// TIA Portal V17 export
// export: Created 2021-12-03T08:13:14.6576163Z, ExportSetting WithDefaults, DisplayName Totally Integrated Automation Portal, DisplayVersion V17, DisplayName TIA Portal Openness, DisplayVersion V17, DisplayName TIA Portal Version Control Interface, DisplayVersion V17, DisplayName STEP 7 Professional, DisplayVersion V17, DisplayName STEP 7 Safety, DisplayVersion V17, DisplayName WinCC Advanced, DisplayVersion V17
FUNCTION "FFC_ReadInputs" : Void   // FC50, F_FBD
VERSION : 0.1
// stored: AutoNumber false, IsIECCheckEnabled false, UDAEnableTagReadback false
BEGIN

REGION Network 2: Консоль ускорителя канал 1
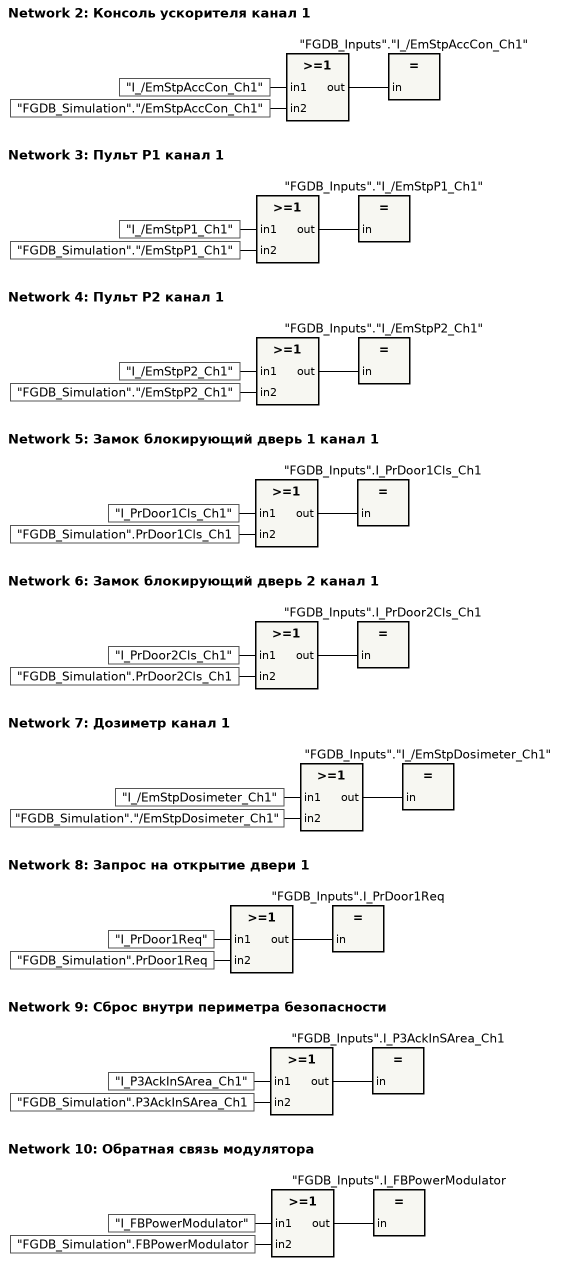
   "FGDB_Inputs"."I_/EmStpAccCon_Ch1" := "I_/EmStpAccCon_Ch1" OR "FGDB_Simulation"."/EmStpAccCon_Ch1";
END_REGION

REGION Network 3: Пульт Р1 канал 1
   "FGDB_Inputs"."I_/EmStpP1_Ch1" := "I_/EmStpP1_Ch1" OR "FGDB_Simulation"."/EmStpP1_Ch1";
END_REGION

REGION Network 4: Пульт Р2 канал 1
   "FGDB_Inputs"."I_/EmStpP2_Ch1" := "I_/EmStpP2_Ch1" OR "FGDB_Simulation"."/EmStpP2_Ch1";
END_REGION

REGION Network 5: Замок блокирующий дверь 1 канал 1
   "FGDB_Inputs".I_PrDoor1Cls_Ch1 := "I_PrDoor1Cls_Ch1" OR "FGDB_Simulation".PrDoor1Cls_Ch1;
END_REGION

REGION Network 6: Замок блокирующий дверь 2 канал 1
   "FGDB_Inputs".I_PrDoor2Cls_Ch1 := "I_PrDoor2Cls_Ch1" OR "FGDB_Simulation".PrDoor2Cls_Ch1;
END_REGION

REGION Network 7: Дозиметр канал 1
   "FGDB_Inputs"."I_/EmStpDosimeter_Ch1" := "I_/EmStpDosimeter_Ch1" OR "FGDB_Simulation"."/EmStpDosimeter_Ch1";
END_REGION

REGION Network 8: Запрос на открытие двери 1
   "FGDB_Inputs".I_PrDoor1Req := "I_PrDoor1Req" OR "FGDB_Simulation".PrDoor1Req;
END_REGION

REGION Network 9: Сброс внутри периметра безопасности
   "FGDB_Inputs".I_P3AckInSArea_Ch1 := "I_P3AckInSArea_Ch1" OR "FGDB_Simulation".P3AckInSArea_Ch1;
END_REGION

REGION Network 10: Обратная связь модулятора
   "FGDB_Inputs".I_FBPowerModulator := "I_FBPowerModulator" OR "FGDB_Simulation".FBPowerModulator;
END_REGION

REGION Network 11: Обратная связь частотного преобразователя
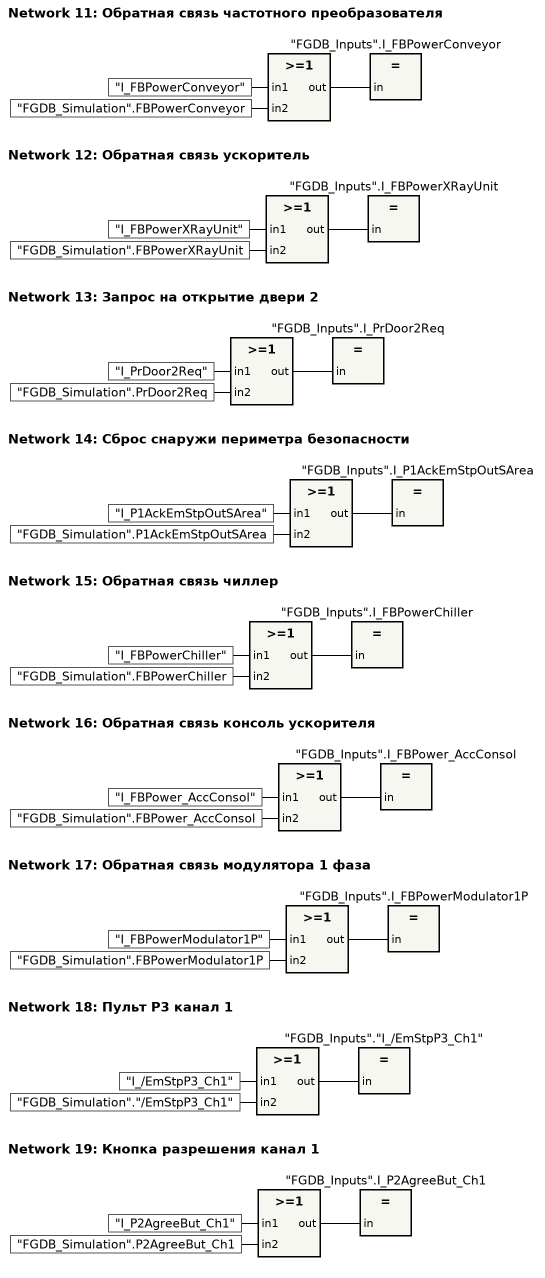
   "FGDB_Inputs".I_FBPowerConveyor := "I_FBPowerConveyor" OR "FGDB_Simulation".FBPowerConveyor;
END_REGION

REGION Network 12: Обратная связь ускоритель
   "FGDB_Inputs".I_FBPowerXRayUnit := "I_FBPowerXRayUnit" OR "FGDB_Simulation".FBPowerXRayUnit;
END_REGION

REGION Network 13: Запрос на открытие двери 2
   "FGDB_Inputs".I_PrDoor2Req := "I_PrDoor2Req" OR "FGDB_Simulation".PrDoor2Req;
END_REGION

REGION Network 14: Сброс снаружи периметра безопасности
   "FGDB_Inputs".I_P1AckEmStpOutSArea := "I_P1AckEmStpOutSArea" OR "FGDB_Simulation".P1AckEmStpOutSArea;
END_REGION

REGION Network 15: Обратная связь чиллер
   "FGDB_Inputs".I_FBPowerChiller := "I_FBPowerChiller" OR "FGDB_Simulation".FBPowerChiller;
END_REGION

REGION Network 16: Обратная связь консоль ускорителя
   "FGDB_Inputs".I_FBPower_AccConsol := "I_FBPower_AccConsol" OR "FGDB_Simulation".FBPower_AccConsol;
END_REGION

REGION Network 17: Обратная связь модулятора 1 фаза
   "FGDB_Inputs".I_FBPowerModulator1P := "I_FBPowerModulator1P" OR "FGDB_Simulation".FBPowerModulator1P;
END_REGION

REGION Network 18: Пульт P3 канал 1
   "FGDB_Inputs"."I_/EmStpP3_Ch1" := "I_/EmStpP3_Ch1" OR "FGDB_Simulation"."/EmStpP3_Ch1";
END_REGION

REGION Network 19: Кнопка разрешения канал 1
   "FGDB_Inputs".I_P2AgreeBut_Ch1 := "I_P2AgreeBut_Ch1" OR "FGDB_Simulation".P2AgreeBut_Ch1;
END_REGION

REGION Network 20: Главный ключ разрешения канал 1
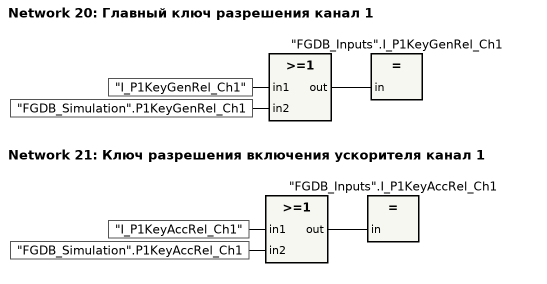
   "FGDB_Inputs".I_P1KeyGenRel_Ch1 := "I_P1KeyGenRel_Ch1" OR "FGDB_Simulation".P1KeyGenRel_Ch1;
END_REGION

REGION Network 21: Ключ разрешения включения ускорителя канал 1
   "FGDB_Inputs".I_P1KeyAccRel_Ch1 := "I_P1KeyAccRel_Ch1" OR "FGDB_Simulation".P1KeyAccRel_Ch1;
END_REGION
END_FUNCTION
